//     SoftDrive 8/Data Pointer/OutputPointer1 <-> Outputs/SoftDriveOutput
//   NC-Task 1 SAF/Axes/Mover Axis 9 <-> TcCOM Objects/XtsProcessingUnit 1/Mover 9
//     SoftDrive 9/Data Pointer/InputPointer1 <-> Inputs/SoftDriveInput
//     SoftDrive 9/Data Pointer/OutputPointer1 <-> Outputs/SoftDriveOutput
//   Test_XTS/Test_XTS Instance <-> NC-Task 1 SAF/Axes/Asse 12
//     PlcTask Inputs/GVL.Asse_Reale.NcToPlc <-> Outputs/ToPlc
//     PlcTask Outputs/GVL.Asse_Reale.PlcToNc <-> Inputs/FromPlc
//   Test_XTS/Test_XTS Instance <-> NC-Task 1 SAF/Axes/Mover Axis 1
//     PlcTask Inputs/GVL.Mover[0].NcToPlc <-> Outputs/ToPlc
//     PlcTask Outputs/GVL.Mover[0].PlcToNc <-> Inputs/FromPlc
//   Test_XTS/Test_XTS Instance <-> NC-Task 1 SAF/Axes/Mover Axis 10
//     PlcTask Inputs/GVL.Mover[9].NcToPlc <-> Outputs/ToPlc
//     PlcTask Outputs/GVL.Mover[9].PlcToNc <-> Inputs/FromPlc
//   Test_XTS/Test_XTS Instance <-> NC-Task 1 SAF/Axes/Mover Axis 2
//     PlcTask Inputs/GVL.Mover[1].NcToPlc <-> Outputs/ToPlc
//     PlcTask Outputs/GVL.Mover[1].PlcToNc <-> Inputs/FromPlc
//   Test_XTS/Test_XTS Instance <-> NC-Task 1 SAF/Axes/Mover Axis 3
//     PlcTask Inputs/GVL.Mover[2].NcToPlc <-> Outputs/ToPlc
//     PlcTask Outputs/GVL.Mover[2].PlcToNc <-> Inputs/FromPlc
//   Test_XTS/Test_XTS Instance <-> NC-Task 1 SAF/Axes/Mover Axis 4
//     PlcTask Inputs/GVL.Mover[3].NcToPlc <-> Outputs/ToPlc
//     PlcTask Outputs/GVL.Mover[3].PlcToNc <-> Inputs/FromPlc
//   Test_XTS/Test_XTS Instance <-> NC-Task 1 SAF/Axes/Mover Axis 5
//     PlcTask Inputs/GVL.Mover[4].NcToPlc <-> Outputs/ToPlc
//     PlcTask Outputs/GVL.Mover[4].PlcToNc <-> Inputs/FromPlc
//   Test_XTS/Test_XTS Instance <-> NC-Task 1 SAF/Axes/Mover Axis 6
//     PlcTask Inputs/GVL.Mover[5].NcToPlc <-> Outputs/ToPlc
//     PlcTask Outputs/GVL.Mover[5].PlcToNc <-> Inputs/FromPlc
//   Test_XTS/Test_XTS Instance <-> NC-Task 1 SAF/Axes/Mover Axis 7
//     PlcTask Inputs/GVL.Mover[6].NcToPlc <-> Outputs/ToPlc
//     PlcTask Outputs/GVL.Mover[6].PlcToNc <-> Inputs/FromPlc
//   Test_XTS/Test_XTS Instance <-> NC-Task 1 SAF/Axes/Mover Axis 8
//     PlcTask Inputs/GVL.Mover[7].NcToPlc <-> Outputs/ToPlc
//     PlcTask Outputs/GVL.Mover[7].PlcToNc <-> Inputs/FromPlc
//   Test_XTS/Test_XTS Instance <-> NC-Task 1 SAF/Axes/Mover Axis 9
//     PlcTask Inputs/GVL.Mover[8].NcToPlc <-> Outputs/ToPlc
//     PlcTask Outputs/GVL.Mover[8].PlcToNc <-> Inputs/FromPlc

CONFIGURATION Test_XTS
    RESOURCE PLC ON TwinCAT3
        TASK PlcTask(INTERVAL := T#10ms, PRIORITY := 21);
        PROGRAM MAIN WITH PlcTask : MAIN;
    END_RESOURCE
END_CONFIGURATION

// ---- GVLs/GVL.TcGVL
{attribute 'qualified_only'}
VAR_GLOBAL

	Mover			:	ARRAY[0..9] OF AXIS_REF;
	
	Asse_Reale		: Axis_ref;
	Asse_Virtuale	: Axis_ref;

END_VAR

// ---- POUs/MAIN.TcPOU
PROGRAM MAIN
VAR
END_VAR

END_PROGRAM
